// TIA Portal V19 export
TYPE "LEXCHANGETRAY_typeTrayStatus"
// stored: Access Published
   STRUCT
      cellsStatus : Int;   // 0: 空盘 1：满盘
      contraintStatus : Int;   // 0:已拘束 1: 解拘束中 2：已解束 3：拘束中
   END_STRUCT;
END_TYPE
